Staubli VAL3: txt_rd1.pgx

public program txt_rd1()
  local num l_ntest
  local num l_n
  local num l_mark
  local bool l_jtest
begin
  //  l_ntest=$fileOpen("test.txt","r")
  //  //  直接更改数量，注意point及sstring要与其一致
  //  //  for l_n=0 to 1
  //  //    $fileGet(l_ntest,sString[l_n],1)
  //  //    if sString[l_n]!=""
  //  //      call stringtopoint(sString[l_n],l_n)
  //  //    endIf
  //  //  endFor
  //  ///////初始化
  //  l_n=0
  //  //  while size(sString)>1
  //  //    $ddel(sString,size(sString)-1)
  //  //  endWhile
  //  //  while size(pfrmCad)>1
  //  //    $ddel(pfrmCad,size(pfrmCad)-1)
  //  //  endWhile
  //  //  while size(jCad)>1
  //  //    $ddel(jCad,size(jCad)-1)
  //  //  endWhile
  //  ///////////////
  //  //  popUpMsg("已经开始读点，请稍等...")
  //  do
  //    if l_n!=0
  //      $dins(sString,l_n)
  //      $dins(pfrmCad,l_n)
  //    endIf
  //    $fileGet(l_ntest,sString[l_n],1)
  //    if sString[l_n]!=""
  //      call stringtopoint(sString[l_n],l_n)
  //    else
  //    endIf
  //    l_n=l_n+1
  //  until sString[l_n-1]==""
  //  $ddel(sString,size(sString)-1)
  //  $ddel(pfrmCad,size(pfrmCad)-1)
  //  delay(0.1)
  //  nScrPts=size(pfrmCad)
  //  call hmi_refreshmain()
  //  popUpMsg("读取完毕")
  //  $fileClose(l_ntest)
  //  //读取参考系中的点
  //  //  call jCadClean()
  //  //清空jcad
  //  //  nTotalPoints=size(pfrmCad)
  //  //  for l_mark=1 to nTotalPoints-1 step 1
  //  //    $dins(jCad,l_mark)
  //  //  endFor
  //  //  for l_mark=0 to size(pfrmCad)-1 step 1
  //  //    l_jtest=pointToJoint(tTool,jConfig,pfrmCad[l_mark],jReal)
  //  //    if l_jtest==false
  //  //      popUpMsg("point is wrong")
  //  //      return
  //  //    else
  //  //      jCad[l_mark]=jReal
  //  //      // jCad[nTotalPoints-1]=jHome
  //  //      //      $dins(jCad,nTotalPoints)
  //  //      ////      nScrPts=nTotalPoints
  //  //      //      nTotalPoints=nTotalPoints+1
  //  //      delay(0)
  //  //    endIf
  //  //  endFor
  //  //   $ddel(jCad,size(jCad))
  //  bfnshint=true
  //  //将pfrmcad逐个转化成jcad的joint点。
  //  /////////////////////////////////////
  //  /////////////////////////////////////
  //  //        call stringToJoints(CmdBuffer[nReadPt],jReal)
  //  //        if bRealM==true
  //  //          //for realtime synchronous movement
  //  //        else
  //  //          //for initialize all points firstly
  //  //          //not realtime synchronous movement
  //  //          nTotalPoints=nTotalPoints+1
  //  //          $dins(jCad,nTotalPoints-1)
  //  //          jCad[nTotalPoints-1]=jReal
  //  //
  //  //          nScrPts=nTotalPoints
  //  //          call hmi_refreshmain()
  //  //        endIf
  //  //      endIf
end
